TYPE AX5000_S_0201 :
STRUCT
	Motor_warning_temperature:UINT;
END_STRUCT
END_TYPE

(* stored: Version 1.1.0.1, ProductVersion 3.1.4024.3
   DUT AX5000_S_0201: Id {f406a21a-4842-48bc-9a05-14acd07a90ab} *)
